{attribute 'linkalways'}
{attribute 'hide_all_locals'}
FUNCTION_BLOCK ValueUint EXTENDS ValueUintRead IMPLEMENTS Value
VAR
END_VAR

METHOD SetFromType : BOOL
VAR_INPUT
	source : __SYSTEM.AnyType;
END_VAR
SetFromType := ConvertAnyType(source, thisAnyType);
END_METHOD

METHOD SetFromString : BOOL
VAR_INPUT
	value : T_MaxString;
END_VAR
thisValue := STRING_TO_UINT(value);

SetFromString := TRUE;
END_METHOD

METHOD Set : BOOL
VAR_INPUT
	source : ANY;
END_VAR
Set := ConvertAnyType(source, thisAnyType);
END_METHOD

END_FUNCTION_BLOCK

(* stored: Version 1.1.0.1
   POU ValueUint: Id {e76b0894-2abd-46cc-8360-63ac8f9fbed9}, SpecialFunc None
   Method SetFromType: Id {a1152134-cde0-4379-9300-13813343ac78}
   Method SetFromString: Id {c66db27c-8997-4cbe-888a-337e8e06a07f}
   Method Set: Id {7dced064-d0e3-4f8f-aac9-18bbce822e2c} *)
